FUNCTION F_GetElementErrorData : ST_ElementErrorStruct
(**************************************************************************************
 * 	Application		:	BoxControl Framework
 *	Revision		:	$Revision: 404529 $
 *	Revision date	:	$Date: 2018-04-23 08:21:38 +0200 (Mo., 23 Apr 2018) $
 *	Last changed by	:	$Author: b7bolm $
 *	URL				:	$URL: http://almscdc.swisslog.com/repo/SWPD/Development/BoxControlFramework/20_Release/trunk/01_Software/BCF/BCF/JumpStart/20_Product/10_App/13_Elements/10_Lib/10_Conv/10_Functions/F_GetElementErrorData.TcPOU $
 *
 *	Purpose			:	Return element error data
 *
 * ------------------------------------------------------------------------------------
 *	Copyright Swisslog [IP AG], Switzerland. All rights reserved.
 * 
 * ------------------------------------------------------------------------------------
 *	
 * 	Revision History: 
 *
 * 	VERSION			DATE			INITIALS			DESCRIPTION
 *	0.1				01.01.2001		swl					Example
 *
 **************************************************************************************)
VAR_INPUT
	eElementNumber		: E_ElementNumber; // Element number
END_VAR


// Check if element number is valid
IF eElementNumber > E_ElementNumber.E_BEGIN_ELEMENT AND
   eElementNumber < E_ElementNumber.E_END_ELEMENT THEN
  
	// Check reference is valid
	IF __ISVALIDREF(ElementRegistry[eElementNumber].rElementData) THEN
   		// Return error data
   		F_GetElementErrorData := ElementRegistry[eElementNumber].rElementData.ErrorData;
	END_IF
END_IF

END_FUNCTION

(* stored: Version 1.1.0.1, ProductVersion 3.1.4022.12
   POU F_GetElementErrorData: Id {22caf12b-7c50-44f9-b848-34f9695663fd}, SpecialFunc None *)
